Universal Robots URScript: COOK ROUTINE.script

def COOK_ROUTINE_3_4318():
  set_standard_analog_input_domain(0, 1)
  set_standard_analog_input_domain(1, 1)
  set_tool_analog_input_domain(0, 1)
  set_tool_analog_input_domain(1, 1)
  set_analog_outputdomain(0, 0)
  set_analog_outputdomain(1, 0)
  set_tool_voltage(0)
  set_standard_digital_input_action(0, "default")
  set_standard_digital_input_action(1, "default")
  set_standard_digital_input_action(2, "default")
  set_standard_digital_input_action(3, "default")
  set_standard_digital_input_action(4, "default")
  set_standard_digital_input_action(5, "default")
  set_standard_digital_input_action(6, "default")
  set_standard_digital_input_action(7, "default")
  set_tool_digital_input_action(0, "default")
  set_tool_digital_input_action(1, "default")
  set_tcp(p[0.0,0.0,0.0,0.0,0.0,0.0])
  set_payload(0.0)
  set_gravity([0.0, 0.0, 9.82])
  rtde_set_watchdog("speed_slider_mask", 10.0, "ignore")
  def To_Grill():
    movej([0.5955818891525269, -2.0482681433307093, -1.3355329672442835, -3.9537580649005335, -2.227043930684225, -0.6348198095904749], a=1.3962634015954636, v=1.0471975511965976)
    movej([0.5772730631269657, -2.0609714578644205, -1.656070522800409, -3.3718257025431333, -2.288818075318295, -0.6212277678003755], a=1.3962634015954636, v=1.0471975511965976)
    movej([0.6105535626411438, -2.0779054800616663, -1.6419513861285608, -3.3409460226642054, -2.2634719053851526, -0.6004465262042444], a=1.3962634015954636, v=1.0471975511965976)
    movej([0.6164344549179077, -2.0414932409869593, -1.6418078581439417, -3.357230011616842, -2.263496224080221, -0.6004703680621546], a=1.3962634015954636, v=1.0471975511965976)
    movej([0.7006521224975586, -2.0909879843341272, -1.5754206816302698, -3.395378891621725, -2.172079865132467, -0.46093589464296514], a=1.3962634015954636, v=1.0471975511965976)
    movej([0.803208589553833, -2.136280361806051, -1.4548185507403772, -3.478126827870504, -2.0544684568988245, -0.4623497168170374], a=1.3962634015954636, v=1.0471975511965976)
    movej([0.803268551826477, -2.104992214833395, -1.455153767262594, -3.478198830281393, -2.0544326941119593, -0.46237355867494756], a=1.3962634015954636, v=1.0471975511965976)
    movej([0.8234316110610962, -2.133946243916647, -1.4558242003070276, -3.4393861929522913, -2.054420773183004, -0.4619663397418421], a=1.3962634015954636, v=1.0471975511965976)
    movej([0.8232032634673541, -2.047395285350925, -1.2757572874463783, -3.706798564918703, -2.0570130472500807, -0.4637103384831285], a=1.3962634015954636, v=1.0471975511965976)
    movej([1.768154501914978, -1.631885830556051, -2.158698383961813, -1.886695686970846, -1.4170544783221644, 0.08916451036930084], a=1.3962634015954636, v=1.0471975511965976)
    movej([1.698920488357544, -1.7186315695392054, -1.717130486165182, -3.369012180958883, -1.3957536856280726, 0.08905664831399918], a=1.3962634015954636, v=1.0471975511965976, r=0.034)
    movej([1.6414695978164673, -2.134448830281393, -1.0955870787249964, -4.006693188344137, -1.451550308858053, 0.08269265294075012], a=1.3962634015954636, v=1.0471975511965976)
    movej([1.6415128467227351, -2.1380718125712104, -1.1246639610957399, -3.9740336213372043, -1.4513190918711611, 0.08301056531857753], a=1.3962634015954636, v=1.0471975511965976)
    movej([1.6687340958351906, -1.7777729489071357, -1.635101249141698, -3.827226810661165, -1.4343775267001773, 0.10676117266883468], a=1.3962634015954636, v=1.0471975511965976)
    movej([1.6686475276947021, -1.5514896551715296, -1.630866829548971, -4.151597325001852, -1.4342368284808558, 0.10673413425683975], a=1.3962634015954636, v=1.0471975511965976)
  end
  def Flip():
    movej([1.7708683444818067, -1.633851163435109, -1.694508390466396, -3.498378443876027, -1.4127499966032708, 0.08960905186847246], t=4.0)
    movej([1.5200145347853855, -1.7766409967187684, -1.812911925922803, -3.3976649241421377, -1.6551373245800516, -0.0081875678372203], a=1.3962634015954636, v=1.0471975511965976)
    movej([1.5898984670639038, -2.0458744207965296, -1.4941838423358362, -3.3674915472613733, -1.5588062445269983, 0.06704088300466537], a=1.3962634015954636, v=1.0471975511965976)
    movej([1.5445931117401948, -1.9877265190245978, -1.7603055658110618, -2.827502633245121, -1.563780962657038, -0.020626333518274365], t=1.0, r=0.05)
    movej([1.615455985069275, -1.8939154783831995, -2.14213210741152, -1.9066742102252405, -1.4978745619403284, 3.954794374294579E-4], a=1.3962634015954636, v=1.0471975511965976)
    movej([1.61546790599823, -1.6603625456439417, -1.9227336088763636, -1.7480695883380335, -1.4953959623919886, 8.029430755414069E-4], t=1.0, r=0.002)
    movej([1.714249849319458, -1.9193671385394495, -1.730574909840719, -1.0380094687091272, -1.0708583037005823, -1.6973632017718714], t=0.5, r=0.023)
    movej([1.7249850034713745, -1.9206002394305628, -1.8837688604937952, -0.991333309804098, -1.4932649771319788, -3.0518341700183313], t=0.5, r=0.018)
    movej([1.6755198240280151, -1.7474525610553187, -2.0974538961993616, -1.8535931746112269, -1.4033568541156214, -3.145057026539938], t=0.5)
    movej([1.669801937257287, -1.7454374445491254, -1.992464200886463, -2.575965468084575, -1.3978528199829885, -3.1451190747923823], t=1.0, r=0.002)
    movej([1.644454116797123, -1.6363896580902484, -2.103503207574808, -2.614357829083252, -1.4252760733915038, -3.147974516817855], t=0.5, r=0.05)
    movej([1.7033982475304896, -1.512872505744057, -1.9461825269616906, -2.897777558942364, -1.3692764163182662, -3.142745635506468], a=1.3962634015954636, v=1.0471975511965976, r=0.044)
  end
  def Off_Grill():
    movej([1.7708683444818067, -1.633851163435109, -1.694508390466396, -3.498378443876027, -1.4127499966032708, 0.08960905186847246], t=4.0)
    movej([1.5697511827555894, -1.76309865437565, -1.8293898422928336, -3.393125987582662, -1.6171828060832496, 0.024053408432931356], a=1.3962634015954636, v=1.0471975511965976)
    movej([1.6016718558616525, -2.051694190320326, -1.4861723479324578, -3.359402106783701, -1.495819502713628, -3.81396104994991E-4], a=1.3962634015954636, v=1.0471975511965976)
    movej([1.6163551807403564, -1.972938362752096, -1.7829893271075647, -2.8211491743670862, -1.4950006643878382, 9.58738019107841E-5], t=1.0, r=0.05)
    movej([1.615455985069275, -1.8939154783831995, -2.14213210741152, -1.9066742102252405, -1.4978745619403284, 3.954794374294579E-4], a=1.3962634015954636, v=1.0471975511965976)
    movej([1.0606755018234253, -2.1703317801104944, -1.0463584105121058, -3.6301830450641077, -1.793253246937887, -0.20118219057192022], t=1.0, r=0.002)
    movej([1.0611428022384644, -2.414633099232809, -0.5990584532367151, -4.289918367062704, -1.6779754797564905, -0.4587796370135706], t=0.5, r=0.023)
    movej([1.061094880104065, -2.281864945088522, -0.5963061491595667, -4.289954368268148, -1.6779635588275355, -0.4587314764605921], t=0.5, r=0.018)
  end
  def Center():
    movej([1.7708683444818067, -1.633851163435109, -1.694508390466396, -3.498378443876027, -1.4127499966032708, 0.08960905186847246], t=4.0)
    movej([1.6173386573791504, -1.6567462126361292, -1.8543489615069788, -3.541016403828756, -1.544701878224508, 0.08958395570516586], a=1.3962634015954636, v=1.0471975511965976)
    movej([1.6084343252778082, -1.8395915441300144, -1.6343334825985094, -3.5779440057268292, -1.5515307317374365, 0.08312999040883629], t=4.0)
    movej([1.6155039072036743, -1.777961556111471, -1.6061232725726526, -3.7027466932879847, -1.516409699116842, 0.13705609738826752], a=1.3962634015954636, v=1.0471975511965976)
    movej([1.6842317859895555, -2.313261123379471, -0.6499215873561033, -1.80373577014905, 0.8817351596644185, 1.7486982361007044], t=4.0)
    movej([1.6839467589810013, -2.2931935562469974, -0.8694992891572717, -1.6057227943038246, 0.8821748586160109, 1.7510396921112772], a=1.3962634015954636, v=1.0471975511965976)
    movej([1.7134938999343792, -2.292487417934714, -0.861470840133796, -1.638973298644796, 0.8841783084279116, 1.7891629668304174], t=4.0)
    movej([1.7137376196671268, -2.3042890812618317, -0.7007587128845643, -1.7867304861246396, 0.8838281517828301, 1.7873660421819437], a=1.3962634015954636, v=1.0471975511965976)
    movej([1.6006797552108765, -2.070245091115133, -0.7604110876666468, -1.5182479063617151, 1.5861799716949463, 0.11639416962862015], a=1.3962634015954636, v=1.0471975511965976)
    movej([1.531215073597356, -2.2794507840190494, -0.7431855092787512, -1.6806811936546246, 2.2498896484060396, -1.5735034079784667], a=1.3962634015954636, v=1.0471975511965976)
    movej([1.5309836461390152, -2.2712405125594355, -0.9078857483329479, -1.5230391690016916, 2.2500805008424276, -1.5716586877214134], a=1.3962634015954636, v=1.0471975511965976)
    movej([1.4605849774807904, -2.307924539599, -0.8423433747292108, -1.6082178425987301, 2.2489101660825632, -1.6625109746335287], t=4.0)
    movej([1.4607340860977254, -2.313853020192788, -0.7328937766459207, -1.712495691893242, 2.248728280967434, -1.6637246251623186], a=1.3962634015954636, v=1.0471975511965976)
    movej([1.604134202003479, -2.020341221486227, -0.7518551985370081, -1.957228962575094, 1.5903666019439697, -2.9874466101275843], a=1.3962634015954636, v=1.0471975511965976)
  end
  $ 1 "Robot Program"
  $ 2 "x≔0"
  global x=0
  $ 3 "y≔0"
  global y=0
  $ 4 "MoveJ"
  $ 5 "Start"
  movej([1.7708683444818067, -1.633851163435109, -1.694508390466396, -3.498378443876027, -1.4127499966032708, 0.08960905186847246], a=1.3962634015954636, v=1.0471975511965976)
  $ 7 "Call To_Grill"
  To_Grill()
  $ 8 "Call Center"
  Center()
  $ 9 "Call Flip"
  Flip()
  $ 10 "Call Center"
  Center()
  $ 11 "Call Off_Grill"
  Off_Grill()
end
